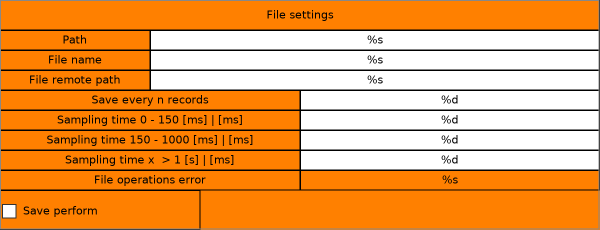
VISUALIZATION vFileSave  // 600x230
VAR_IN_OUT
	fbChamber 	: fbChamber;
	stParams	: stParamsChamber;
END_VAR
    Rectangle (0,190 200x40)
    Rectangle (0,0 600x30), "File settings"
    Rectangle (0,30 150x20), "Path"
    Rectangle (150,30 450x20), "%s", text variable: stParams.sFileDirectory
        OnMouseClick: write the text variable via VisuDialogs.Keypad
    Rectangle (0,50 150x20), "File name"
    Rectangle (150,50 450x20), "%s", text variable: fbChamber.sTestName
        OnMouseClick: write the text variable via VisuDialogs.Keypad
    Rectangle (0,90 300x20), "Save every n records"
    Rectangle (300,90 300x20), "%d", text variable: stParams.iSaveEveryRecords
        OnMouseClick: write the text variable via Default
    Rectangle (0,130 300x20), "Sampling time 150 - 1000 [ms] | [ms]"
    Rectangle (300,130 300x20), "%d", text variable: stParams.iSampleTime0_1
        OnMouseClick: write the text variable via Default
    Rectangle (0,170 300x20), "File operations error"
    Rectangle (300,170 300x20), "%s", text variable: fbChamber.bFileSaveError, text list: ''
    Rectangle (0,150 300x20), "Sampling time x > 1 [s] | [ms]"
    Rectangle (300,150 300x20), "%d", text variable: stParams.iSampleTime1_x
        OnMouseClick: write the text variable via Default
    Checkbox (0,196 200x30), "Save perform", variable: stParams.bSaveToFile
    Rectangle (0,110 300x20), "Sampling time 0 - 150 [ms] | [ms]"
    Rectangle (300,110 300x20), "%d", text variable: stParams.iSampleTime0_150
        OnMouseClick: write the text variable via Default
    Rectangle (0,70 150x20), "File remote path"
    Rectangle (150,70 450x20), "%s", text variable: stParams.sFileCopyLocation
        OnMouseClick: write the text variable via Edit
END_VISUALIZATION

(* stored: Version 1.1.0.1, ProductVersion 3.1.4024.12
   Visu vFileSave: Id {ec74ecaf-bad0-48bd-867c-a1b30ea91094} *)
